FUNCTION_BLOCK EQUIP_ExitConveyor (* Composite Function Block Type *)
  (* Standard: 61499-2 *)
  (* Version 0.0, 08/01/2026, Schneider Electric, template *)
  PACKAGE Main;
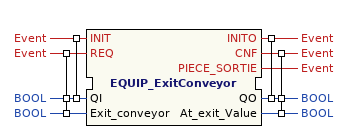
  EVENT_INPUT
    INIT WITH QI; (* Initialization Request *)
    REQ WITH QI, Exit_conveyor; (* Normal Execution Request *)
  END_EVENT
  EVENT_OUTPUT
    INITO WITH QO; (* Initialization Confirm *)
    CNF WITH QO, At_exit_Value; (* Execution Confirmation *)
    PIECE_SORTIE;
  END_EVENT
  VAR_INPUT
    QI : BOOL; (* Input event qualifier *)
    Exit_conveyor : BOOL;
  END_VAR
  VAR_OUTPUT
    QO : BOOL; (* Output event qualifier *)
    At_exit_Value : BOOL; (* Valeur actuelle du capteur At_exit *)
  END_VAR
  FBS
    ReadAtExit : SYMLINKMULTIVARDST_1559B0FF8170C9BA0(NAME1 := 'At_exit'); {SET_ATTRIBUTE(Configuration.GenericFBType.InterfaceParams, Runtime.System#I:=1;VALUE${I$}:BOOL)}
    WriteAtExit : SYMLINKMULTIVARSRC_1559B0FF8170C9BA0(NAME1 := 'Exit_conveyor'); {SET_ATTRIBUTE(Configuration.GenericFBType.InterfaceParams, Runtime.System#I:=1;VALUE${I$}:BOOL)}
    FallingTrig : E_F_TRIG;
  END_FBS
  EVENT_CONNECTIONS
    INIT TO ReadAtExit.INIT;
    REQ TO ReadAtExit.REQ;
    WriteAtExit.INITO TO INITO;
    WriteAtExit.CNF TO CNF;
    ReadAtExit.INITO TO WriteAtExit.INIT;
    ReadAtExit.CNF TO WriteAtExit.REQ;
    ReadAtExit.CNF TO FallingTrig.EI;
    FallingTrig.EO TO PIECE_SORTIE;
  END_CONNECTIONS
  DATA_CONNECTIONS
    WriteAtExit.QO TO QO;
    Exit_conveyor TO WriteAtExit.VALUE1;
    QI TO ReadAtExit.QI;
    ReadAtExit.QO TO WriteAtExit.QI;
    ReadAtExit.VALUE1 TO FallingTrig.QI;
    ReadAtExit.VALUE1 TO At_exit_Value;
  END_CONNECTIONS
END_FUNCTION_BLOCK
